{attribute 'linkalways'} 
{attribute 'no_explicit_call' := 'This FB is a CLASS and must be accessed using methods or properties'}
{attribute 'enable_dynamic_creation'}
FUNCTION_BLOCK FINAL MIN_INT EXTENDS Node
VAR
	in1 : _INT(0);
	in2 : _INT(0);
	out : _INT(0);
END_VAR

METHOD PUBLIC Clone : I_Node
VAR
	pNode : POINTER TO MIN_INT;
END_VAR
pNode := __NEW(MIN_INT);
Clone := pNode^;
END_METHOD

METHOD FB_init : BOOL
VAR_INPUT
	bInitRetains : BOOL; // if TRUE, the retain variables are initialized (warm start / cold start)
	bInCopyCode : BOOL;  // if TRUE, the instance afterwards gets moved into the copy code (online change)
END_VAR
AddInput('in1',THIS^.in1);
AddInput('in2',THIS^.in2);
AddOutput('out', THIS^.out);
END_METHOD

METHOD PROTECTED OnExecute
VAR
END_VAR
out.Value := MIN(in1.Value, in2.Value);
END_METHOD

END_FUNCTION_BLOCK

(* stored: Version 1.1.0.1, ProductVersion 3.1.4024.15
   POU MIN_INT: Id {b350437d-f0fc-49c8-98bf-c8e3f5de5933}, SpecialFunc None
   Folder Constructor: Id {793b9474-1424-4b61-becf-f7668c6db6a5}
   Method Clone: Id {884e2da7-ec56-491b-bc99-5a13366d27fc}
   Method FB_init: Id {2cd3bafc-5bd8-48b7-b9ce-1bc7befa122b}
   Method OnExecute: Id {3df78958-74c9-478a-9a39-8da10022364e} *)
